INTERFACE I_Mover EXTENDS I_MoverPos

METHOD Cyclic : BOOL
VAR_INPUT
END_VAR
END_METHOD

PROPERTY ErrorCode : UDINT
GET
END_GET
END_PROPERTY

PROPERTY Linked : BOOL
GET
END_GET
END_PROPERTY

METHOD SetPosLink : BOOL
VAR_INPUT
	position : I_PosMover;
END_VAR
END_METHOD

PROPERTY State : UDINT
GET
END_GET
SET
END_SET
END_PROPERTY

PROPERTY Step : UDINT
GET
END_GET
END_PROPERTY

METHOD Unlink : BOOL
VAR_INPUT
END_VAR
END_METHOD

METHOD Update : BOOL
VAR_INPUT
END_VAR
END_METHOD

END_INTERFACE

(* stored: Version 1.1.0.1
   Itf I_Mover: Id {88e38cd4-8394-40a2-aa1c-f4649c1e2306}
   Method Cyclic: Id {57530218-a4a1-4d26-b9f0-80ef1595e5ac}
   Property ErrorCode: Id {04cc57bd-f551-47df-b97c-1caa59b3eb19}
   Get Get: Id {93195d7e-270b-4fe8-82a8-91627d30f9e7}
   Property Linked: Id {d2082c7c-f084-4a28-9d8d-9754a6d21e86}
   Get Get: Id {efb52f18-36ac-400e-b9dc-55cdbb74a5b6}
   Method SetPosLink: Id {54a5ad44-1706-4fbc-bcea-7fca19f2bdc4}
   Property State: Id {eb0860e8-01ca-4e58-b300-2ad61efb52d2}
   Get Get: Id {0b64d9ac-fae5-4121-9115-11449e8cdaff}
   Set Set: Id {1f917c3a-54c0-4c85-b30a-9f1389387410}
   Property Step: Id {9da493df-02ec-4a23-afa1-f4d6271b56b6}
   Get Get: Id {f8f74bcd-6b09-4594-aaf4-e5717ab36432}
   Method Unlink: Id {29c21fd2-afc9-4777-b33a-9988cc23f15c}
   Method Update: Id {0fb52271-36e5-43a4-82a0-7b7ce5d9b082} *)
